# EPICS substitutions: streamApp/pluginDb/dataStream.substitutions
# dataStream.substitutions

# ROI Plugin
file NDPluginBase.template
{
	{
	PORT			= "$(IMAGE_NAME):ROI",
	P				= "$(CAM):",
	R				= "$(PORT):",
	ADDR			= "\$(ADDR=0)",
	TIMEOUT			= "\$(TIMEOUT=1)",
	Enable          = "0",
	TSE				= "\$(TSE=-2)",
	NDARRAY_PORT	= "$(CAM_PORT)",
	NDARRAY_ADDR	= "\$(NDARRAY_ADDR=0)",
	}
}
file NDROI.template
{
	{
	PORT			= "$(IMAGE_NAME):ROI",
	P				= "$(CAM):",
	R				= "$(PORT):",
	ADDR			= "\$(ADDR=0)",
	TIMEOUT			= "\$(TIMEOUT=1)",
	}
}

# ColorConvert plugin
file NDPluginBase.template
{
	{
	PORT			= "$(IMAGE_NAME):CC",
	P				= "$(CAM):",
	R				= "$(PORT):",
	ADDR			= "\$(ADDR=0)",
	TIMEOUT			= "\$(TIMEOUT=1)",
	Enable          = "0",
	TSE				= "\$(TSE=-2)",
	NDARRAY_PORT	= "$(CAM_PORT)",
	NDARRAY_ADDR	= "\$(NDARRAY_ADDR=0)",
	}
}
file NDColorConvert.template
{
	{
	P				= "$(CAM):",
	PORT			= "$(IMAGE_NAME):CC",
	R				= "$(PORT):",
	ADDR			= "\$(ADDR=0)",
	TIMEOUT			= "\$(TIMEOUT=1)",
	}
}

# stdArray Plugin
file NDPluginBase.template
{
	{
	PORT			= "$(IMAGE_NAME)",
	P				= "$(CAM):",
	R				= "$(PORT):",
	ADDR			= "\$(ADDR=0)",
	TIMEOUT			= "\$(TIMEOUT=1)",
	Enable          = "1",
	TSE				= "\$(TSE=-2)",
	NDARRAY_PORT	= "$(CAM_PORT)",
	NDARRAY_ADDR	= "\$(NDARRAY_ADDR=0)",
	}
}
file NDStdArrays.template
{
	{
	PORT			= "$(IMAGE_NAME)",
	P				= "$(CAM):",
	R				= "$(PORT):",
	ADDR			= "\$(ADDR=0)",
	TIMEOUT			= "\$(TIMEOUT=1)",
	TYPE		 	= "$(IMAGE_TYPE)",
	FTVL		 	= "$(IMAGE_FTVL)",
	NELEMENTS		= "$(IMAGE_NELM)",
	}
}
